// TIA Portal V20 export
TYPE "UserDiag_typeDevice"
TITLE = UserDiag_typeDevice
   STRUCT
      hardwareId { ExternalAccessible := 'False'; ExternalVisible := 'False'; ExternalWritable := 'False'} : HW_DEVICE := 16#0000;   // Hardware identifier of the device/slave
      number { ExternalAccessible := 'False'; ExternalVisible := 'False'; ExternalWritable := 'False'} : UInt := 0;   // Profinet device number/Profibus address of the slave
      "name" { ExternalAccessible := 'False'; ExternalVisible := 'False'; ExternalWritable := 'False'} : String[50];   // Name of the device/slave
      ipAddress { ExternalAccessible := 'False'; ExternalVisible := 'False'; ExternalWritable := 'False'; S7_SetPoint := 'True'} : IP_V4;   // IP address of the device
      state { ExternalAccessible := 'False'; ExternalVisible := 'False'; ExternalWritable := 'False'} : USInt := 0;   // Status of the device/slave. 1:ok; 2:faulty, 3:lost connection, 4:disabled, 5:problem, 12:was faulty, 13:was lost, 14:was disabled, 15:problem gone
      exists { ExternalAccessible := 'False'; ExternalVisible := 'False'; ExternalWritable := 'False'} : Bool := FALSE;   // TRUE: Device/slave is existing
      configured { ExternalAccessible := 'False'; ExternalVisible := 'False'; ExternalWritable := 'False'} : Bool := FALSE;   // TRUE: Device/slave is configured
      faulty { ExternalAccessible := 'False'; ExternalVisible := 'False'; ExternalWritable := 'False'} : Bool := FALSE;   // TRUE: Device/slave is faulty
      problem { ExternalAccessible := 'False'; ExternalVisible := 'False'; ExternalWritable := 'False'} : Bool := FALSE;   // TRUE: Device/slave has a problem
      disabled { ExternalAccessible := 'False'; ExternalVisible := 'False'; ExternalWritable := 'False'} : Bool := FALSE;   // TRUE: Device/slave is disabled
      error { ExternalAccessible := 'False'; ExternalVisible := 'False'; ExternalWritable := 'False'} : Bool := FALSE;   // TRUE: Error in device/slave
      nextDevice { ExternalAccessible := 'False'; ExternalVisible := 'False'; ExternalWritable := 'False'} : Int;   // device number of next device
      actualConfiguredSlots { ExternalAccessible := 'False'; ExternalVisible := 'False'; ExternalWritable := 'False'} : Int := 0;   // Number of configured slots in the device/slave
      slots { ExternalAccessible := 'False'; ExternalVisible := 'False'; ExternalWritable := 'False'; S7_SetPoint := 'True'} : Array[0.."USERDIAG_SLOTS_PER_DEVICE_UPPER_LIM"] of "UserDiag_typeSlot";   // Slot information of a device/slave
   END_STRUCT;
END_TYPE
